{attribute 'GeneratedUsingTerminal: EL1259-0000-0017'}
{attribute addProperty BoxType "EL1259-0000-0017"}
{attribute addProperty Id "Output_buffer_resetBOOL1Manual_output_stateBOOL1Force_orderBOOL1Enable_manual_operationBOOL1Output_order_counterUSINT1No_of_output_eventsUSINT1"}
{attribute addProperty CRC "2001079251"}
{attribute addProperty Size "6"}
TYPE Ctrl_77460BD3 :
STRUCT
	{attribute addProperty Name "Output_buffer_reset"}
	Output_buffer_reset : BOOL;
	{attribute addProperty Name "Manual_output_state"}
	Manual_output_state : BOOL;
	{attribute addProperty Name "Force_order"}
	Force_order : BOOL;
	{attribute addProperty Name "Enable_manual_operation"}
	Enable_manual_operation : BOOL;
	{attribute addProperty Name "Output_order_counter"}
	Output_order_counter : USINT;
	{attribute addProperty Name "No_of_output_events"}
	No_of_output_events : USINT;
END_STRUCT
END_TYPE

(* stored: Version 1.2.0.0, ProductVersion 3.1.4024.9
   DUT Ctrl_77460BD3: Id {18321de3-6a0a-4de4-a455-5d215f61e27f} *)
